TYPE "UDT_Marking CharToASCII"
VERSION : 0.1
   STRUCT
      "Byte" : Array[0..127] of Byte;
   END_STRUCT;

END_TYPE

